% RSLogix 500 project P4_IVANOVSKI_M.RSS, saved by version 8.30.00.16 %
PROJECT "UNTITLED"    % processor: Bul.1763 MicroLogix 1100 Series B %

PROGRAM FILES
  LAD 2 "MAIN"  7 rungs
  LAD 3 "IO"  8 rungs
  LAD 4 "CONTROLS"  9 rungs
  LAD 5 "STATUS"  9 rungs

DATA FILES
  O0 OUTPUT  4 elements
  I1 INPUT  6 elements
  S2 STATUS  66 elements
  B3 BINARY  2 elements
  T4 TIMER  3 elements
  C5 COUNTER  1 elements
  R6 CONTROL  1 elements
  N7 INTEGER  2 elements
  F8 FLOAT  1 elements

LADDER 2 "MAIN"
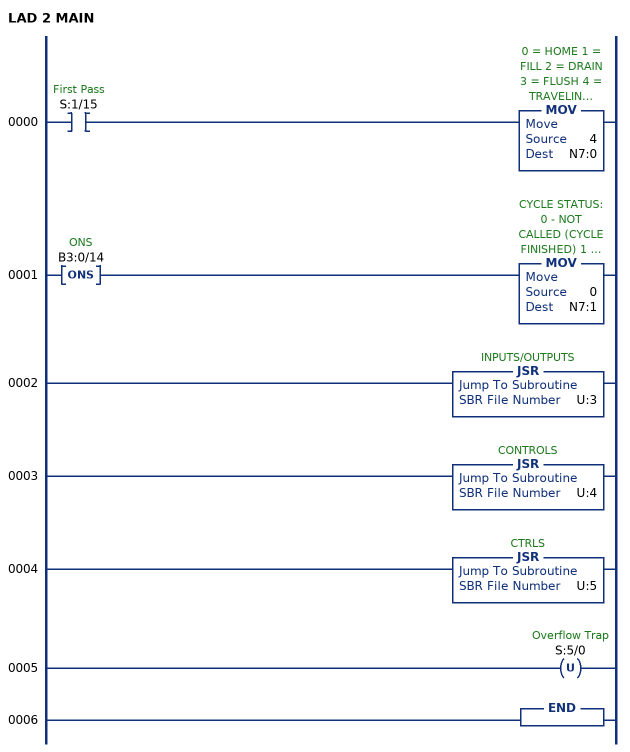
% Rung: 0 %
SOR XIC S:1/15 MOV 4 N7:0 EOR
%   S:1/15  "First Pass" %
%   N7:0  VALVE_POSITION  "0 = HOME 1 = FILL 2 = DRAIN 3 = FLUSH 4 = TRAVELING" %
% Rung: 1 %
SOR ONS B3:0/14 MOV 0 N7:1 EOR
%   B3:0/14  "ONS" %
%   N7:1  "CYCLE STATUS: 0 - NOT CALLED (CYCLE FINISHED) 1 - CALLED" %
% Rung: 2 %
SOR JSR U:3 EOR
%   U:3  "INPUTS/OUTPUTS" %
% Rung: 3 %
SOR JSR U:4 EOR
%   U:4  "CONTROLS" %
% Rung: 4 %
SOR JSR U:5 EOR
%   U:5  "CTRLS" %
% Rung: 5 %
SOR OTU S:5/0 EOR
%   S:5/0  "Overflow Trap" %
% Rung: 6 %
SOR END EOR

LADDER 3 "IO"
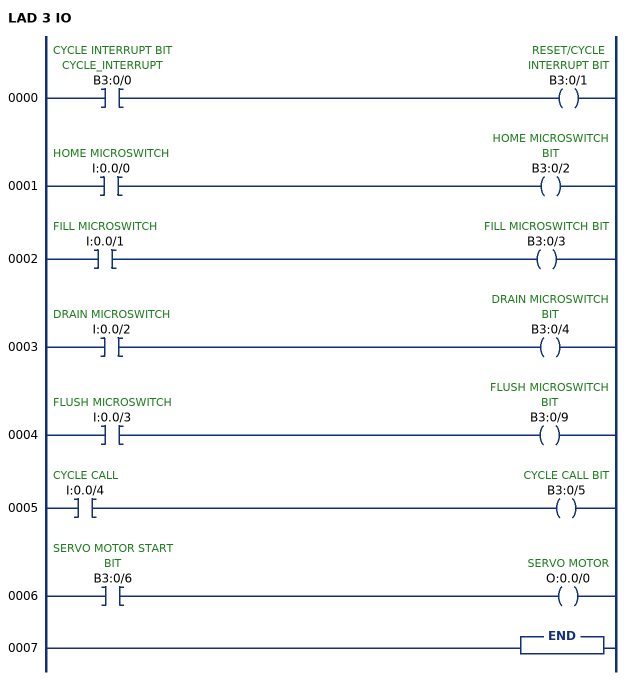
% Rung: 0 %
SOR XIC B3:0/0 OTE B3:0/1 EOR
%   B3:0/0  CYCLE_INTERRUPT  "CYCLE INTERRUPT BIT" %
%   B3:0/1  "RESET/CYCLE INTERRUPT BIT" %
% Rung: 1 %
SOR XIC I:0.0/0 OTE B3:0/2 EOR
%   I:0.0/0  "HOME MICROSWITCH" %
%   B3:0/2  "HOME MICROSWITCH BIT" %
% Rung: 2 %
SOR XIC I:0.0/1 OTE B3:0/3 EOR
%   I:0.0/1  "FILL MICROSWITCH" %
%   B3:0/3  "FILL MICROSWITCH BIT" %
% Rung: 3 %
SOR XIC I:0.0/2 OTE B3:0/4 EOR
%   I:0.0/2  "DRAIN MICROSWITCH" %
%   B3:0/4  "DRAIN MICROSWITCH BIT" %
% Rung: 4 %
SOR XIC I:0.0/3 OTE B3:0/9 EOR
%   I:0.0/3  "FLUSH MICROSWITCH" %
%   B3:0/9  "FLUSH MICROSWITCH BIT" %
% Rung: 5 %
SOR XIC I:0.0/4 OTE B3:0/5 EOR
%   I:0.0/4  "CYCLE CALL" %
%   B3:0/5  "CYCLE CALL BIT" %
% Rung: 6 %
SOR XIC B3:0/6 OTE O:0.0/0 EOR
%   B3:0/6  "SERVO MOTOR START BIT" %
%   O:0.0/0  "SERVO MOTOR" %
% Rung: 7 %
SOR END EOR

LADDER 4 "CONTROLS"
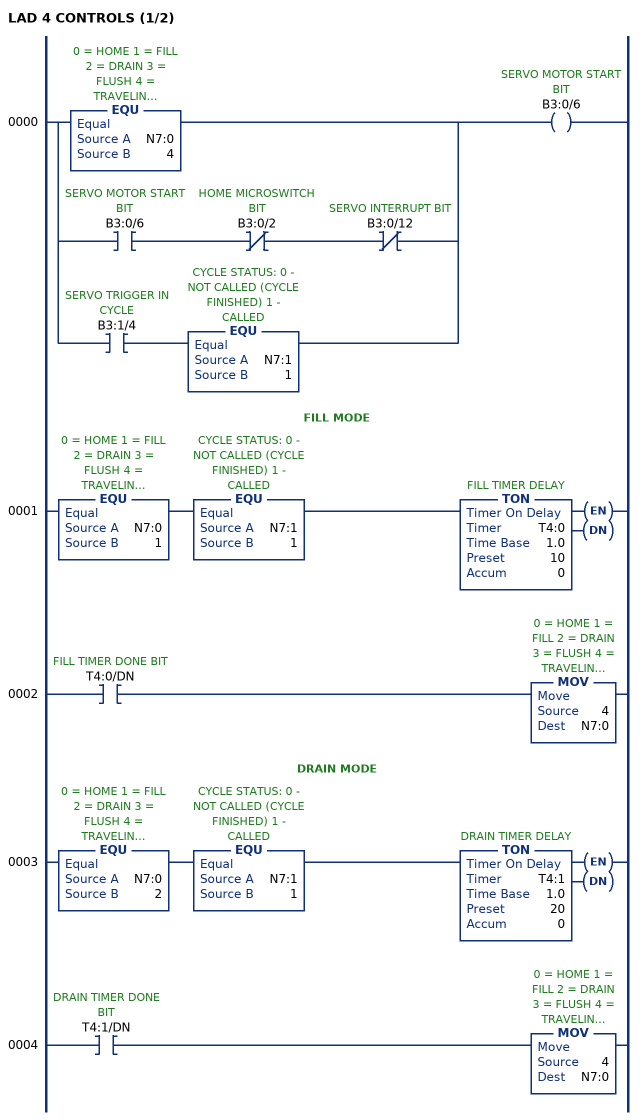
% Rung: 0 %
SOR BST EQU N7:0 4 NXB XIC B3:0/6 XIO B3:0/2 XIO B3:0/12 NXB XIC B3:1/4 EQU N7:1 1 BND OTE B3:0/6 EOR
%   N7:0  VALVE_POSITION  "0 = HOME 1 = FILL 2 = DRAIN 3 = FLUSH 4 = TRAVELING" %
%   B3:0/6  "SERVO MOTOR START BIT" %
%   B3:0/2  "HOME MICROSWITCH BIT" %
%   B3:0/12  "SERVO INTERRUPT BIT" %
%   B3:1/4  "SERVO TRIGGER IN CYCLE" %
%   N7:1  "CYCLE STATUS: 0 - NOT CALLED (CYCLE FINISHED) 1 - CALLED" %
% Rung: 1 %
% TITLE: FILL MODE %
SOR EQU N7:0 1 EQU N7:1 1 TON T4:0 1.0 10 0 EOR
%   N7:0  VALVE_POSITION  "0 = HOME 1 = FILL 2 = DRAIN 3 = FLUSH 4 = TRAVELING" %
%   N7:1  "CYCLE STATUS: 0 - NOT CALLED (CYCLE FINISHED) 1 - CALLED" %
%   T4:0  "FILL TIMER DELAY" %
% Rung: 2 %
SOR XIC T4:0/DN MOV 4 N7:0 EOR
%   T4:0/DN  "FILL TIMER DONE BIT" %
%   N7:0  VALVE_POSITION  "0 = HOME 1 = FILL 2 = DRAIN 3 = FLUSH 4 = TRAVELING" %
% Rung: 3 %
% TITLE: DRAIN MODE %
SOR EQU N7:0 2 EQU N7:1 1 TON T4:1 1.0 20 0 EOR
%   N7:0  VALVE_POSITION  "0 = HOME 1 = FILL 2 = DRAIN 3 = FLUSH 4 = TRAVELING" %
%   N7:1  "CYCLE STATUS: 0 - NOT CALLED (CYCLE FINISHED) 1 - CALLED" %
%   T4:1  "DRAIN TIMER DELAY" %
% Rung: 4 %
SOR XIC T4:1/DN MOV 4 N7:0 EOR
%   T4:1/DN  "DRAIN TIMER DONE BIT" %
%   N7:0  VALVE_POSITION  "0 = HOME 1 = FILL 2 = DRAIN 3 = FLUSH 4 = TRAVELING" %

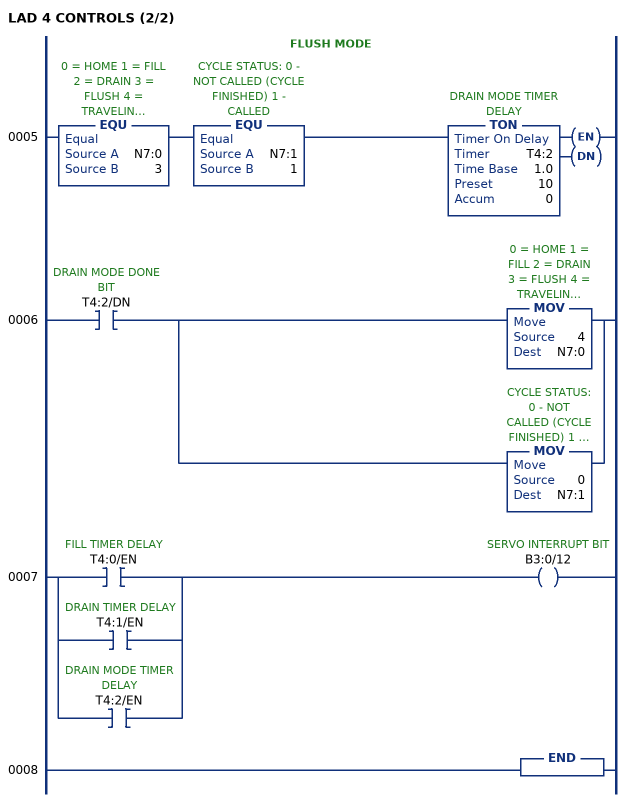
% Rung: 5 %
% TITLE: FLUSH MODE %
SOR EQU N7:0 3 EQU N7:1 1 TON T4:2 1.0 10 0 EOR
%   N7:0  VALVE_POSITION  "0 = HOME 1 = FILL 2 = DRAIN 3 = FLUSH 4 = TRAVELING" %
%   N7:1  "CYCLE STATUS: 0 - NOT CALLED (CYCLE FINISHED) 1 - CALLED" %
%   T4:2  "DRAIN MODE TIMER DELAY" %
% Rung: 6 %
SOR XIC T4:2/DN BST MOV 4 N7:0 NXB MOV 0 N7:1 BND EOR
%   T4:2/DN  "DRAIN MODE DONE BIT" %
%   N7:0  VALVE_POSITION  "0 = HOME 1 = FILL 2 = DRAIN 3 = FLUSH 4 = TRAVELING" %
%   N7:1  "CYCLE STATUS: 0 - NOT CALLED (CYCLE FINISHED) 1 - CALLED" %
% Rung: 7 %
SOR BST XIC T4:0/EN NXB XIC T4:1/EN NXB XIC T4:2/EN BND OTE B3:0/12 EOR
%   T4:0  "FILL TIMER DELAY" %
%   T4:1  "DRAIN TIMER DELAY" %
%   T4:2  "DRAIN MODE TIMER DELAY" %
%   B3:0/12  "SERVO INTERRUPT BIT" %
% Rung: 8 %
SOR END EOR

LADDER 5 "STATUS"
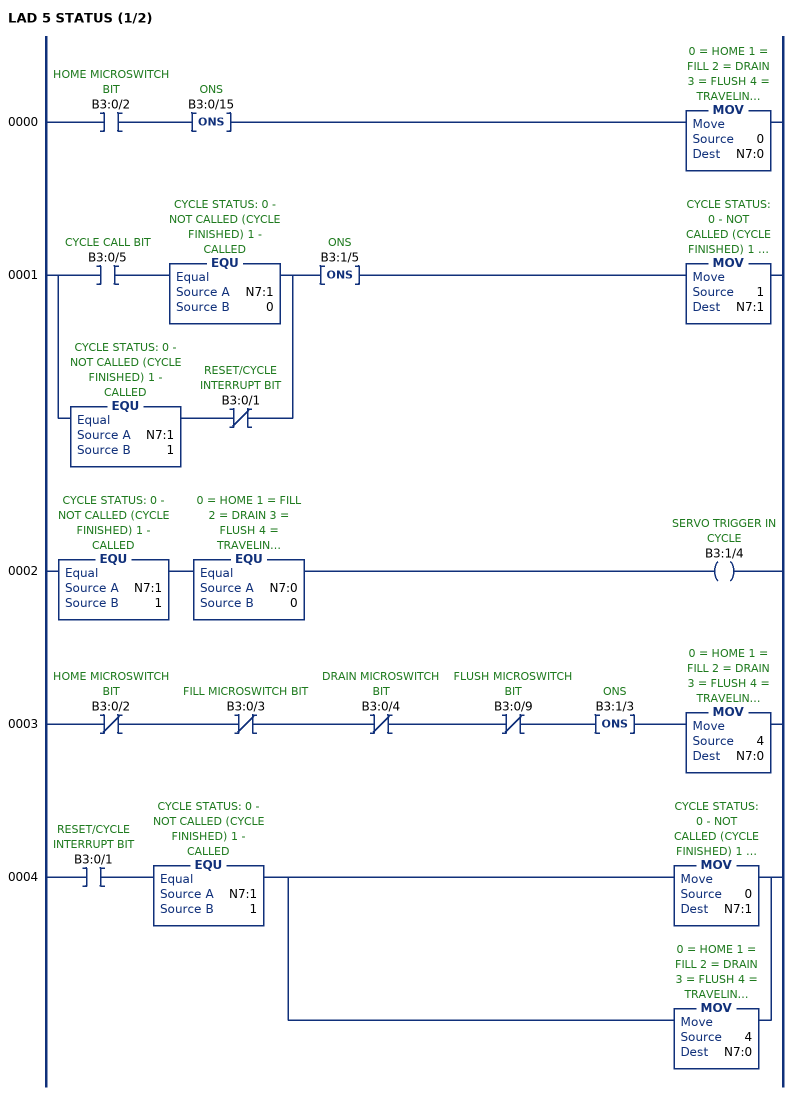
% Rung: 0 %
SOR XIC B3:0/2 ONS B3:0/15 MOV 0 N7:0 EOR
%   B3:0/2  "HOME MICROSWITCH BIT" %
%   B3:0/15  "ONS" %
%   N7:0  VALVE_POSITION  "0 = HOME 1 = FILL 2 = DRAIN 3 = FLUSH 4 = TRAVELING" %
% Rung: 1 %
SOR BST XIC B3:0/5 EQU N7:1 0 NXB EQU N7:1 1 XIO B3:0/1 BND ONS B3:1/5 MOV 1 N7:1 EOR
%   B3:0/5  "CYCLE CALL BIT" %
%   N7:1  "CYCLE STATUS: 0 - NOT CALLED (CYCLE FINISHED) 1 - CALLED" %
%   B3:0/1  "RESET/CYCLE INTERRUPT BIT" %
%   B3:1/5  "ONS" %
% Rung: 2 %
SOR EQU N7:1 1 EQU N7:0 0 OTE B3:1/4 EOR
%   N7:1  "CYCLE STATUS: 0 - NOT CALLED (CYCLE FINISHED) 1 - CALLED" %
%   N7:0  VALVE_POSITION  "0 = HOME 1 = FILL 2 = DRAIN 3 = FLUSH 4 = TRAVELING" %
%   B3:1/4  "SERVO TRIGGER IN CYCLE" %
% Rung: 3 %
SOR XIO B3:0/2 XIO B3:0/3 XIO B3:0/4 XIO B3:0/9 ONS B3:1/3 MOV 4 N7:0 EOR
%   B3:0/2  "HOME MICROSWITCH BIT" %
%   B3:0/3  "FILL MICROSWITCH BIT" %
%   B3:0/4  "DRAIN MICROSWITCH BIT" %
%   B3:0/9  "FLUSH MICROSWITCH BIT" %
%   B3:1/3  "ONS" %
%   N7:0  VALVE_POSITION  "0 = HOME 1 = FILL 2 = DRAIN 3 = FLUSH 4 = TRAVELING" %
% Rung: 4 %
SOR XIC B3:0/1 EQU N7:1 1 BST MOV 0 N7:1 NXB MOV 4 N7:0 BND EOR
%   B3:0/1  "RESET/CYCLE INTERRUPT BIT" %
%   N7:1  "CYCLE STATUS: 0 - NOT CALLED (CYCLE FINISHED) 1 - CALLED" %
%   N7:0  VALVE_POSITION  "0 = HOME 1 = FILL 2 = DRAIN 3 = FLUSH 4 = TRAVELING" %

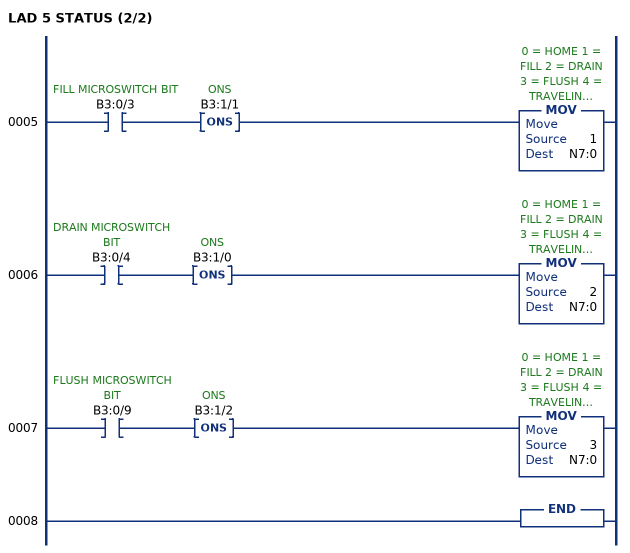
% Rung: 5 %
SOR XIC B3:0/3 ONS B3:1/1 MOV 1 N7:0 EOR
%   B3:0/3  "FILL MICROSWITCH BIT" %
%   B3:1/1  "ONS" %
%   N7:0  VALVE_POSITION  "0 = HOME 1 = FILL 2 = DRAIN 3 = FLUSH 4 = TRAVELING" %
% Rung: 6 %
SOR XIC B3:0/4 ONS B3:1/0 MOV 2 N7:0 EOR
%   B3:0/4  "DRAIN MICROSWITCH BIT" %
%   B3:1/0  "ONS" %
%   N7:0  VALVE_POSITION  "0 = HOME 1 = FILL 2 = DRAIN 3 = FLUSH 4 = TRAVELING" %
% Rung: 7 %
SOR XIC B3:0/9 ONS B3:1/2 MOV 3 N7:0 EOR
%   B3:0/9  "FLUSH MICROSWITCH BIT" %
%   B3:1/2  "ONS" %
%   N7:0  VALVE_POSITION  "0 = HOME 1 = FILL 2 = DRAIN 3 = FLUSH 4 = TRAVELING" %
% Rung: 8 %
SOR END EOR

OTHER DOCUMENTED ADDRESSES
  B3:0/7  "VALVE POSITION BIT"
  B3:0/8  "SERVO TRIGGER START BIT"
  B3:0/10  "ONS"
  B3:0/11  "CYCLE START BIT"
  T4:0.ACC  "FILL TIMER ACCUMULATION BIT"
  T4:0/TT  "FILL TIMER TT BIT"

DATA TABLE (non-zero values as saved)
DATA T4
% .PRE .ACC %
% T4:0 % 10 0
% T4:1 % 20 0
% T4:2 % 10 0
